FUNCTION_BLOCK InputCompressor (* Basic Function Block Type *)
  (* Standard: 61499-2 *)
  (* Version 0.0, 11/1/2016, Dmitry, nxtControl GmbH, Template *)
  PACKAGE Main;
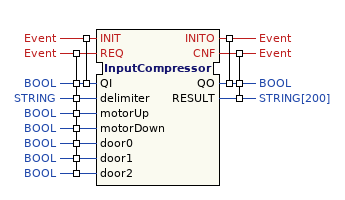
  EVENT_INPUT
    INIT WITH QI; (* Initialization Request *)
    REQ WITH QI, delimiter, motorUp, motorDown, door0, door1, door2; (* Normal Execution Request *)
  END_EVENT
  EVENT_OUTPUT
    INITO WITH QO; (* Initialization Confirm *)
    CNF WITH QO, RESULT; (* Execution Confirmation *)
  END_EVENT
  VAR_INPUT
    QI : BOOL; (* Input event qualifier *)
    delimiter : STRING;
    motorUp : BOOL;
    motorDown : BOOL;
    door0 : BOOL;
    door1 : BOOL;
    door2 : BOOL;
  END_VAR
  VAR_OUTPUT
    QO : BOOL; (* Output event qualifier *)
    RESULT : STRING[200];
  END_VAR
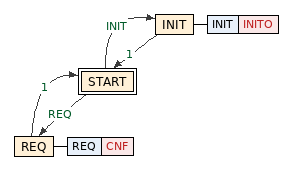
  EC_STATES
    START; (* Initial State *)
    INIT : INIT -> INITO; (* Initialization *)
    REQ : REQ -> CNF; (* Normal execution *)
  END_STATES
  EC_TRANSITIONS
    START TO INIT := INIT;
    INIT TO START := 1;
    START TO REQ := REQ;
    REQ TO START := 1;
  END_TRANSITIONS
  ALGORITHM INIT IN ST: (* Initialization algorithm *)
QO := TRUE;
  END_ALGORITHM
  ALGORITHM REQ IN ST: (* Normally executed algorithm *)
RESULT :=
CONCAT(
  CONCAT(
    BOOL_TO_STRING(motorUp), delimiter,
    BOOL_TO_STRING(motorDown), delimiter,
    BOOL_TO_STRING(door0), delimiter
  ),
  CONCAT(
    BOOL_TO_STRING(door1), delimiter,
    BOOL_TO_STRING(door2), delimiter
  ),
  "$N");
  END_ALGORITHM
END_FUNCTION_BLOCK
